// TIA Portal V19 export
DATA_BLOCK "Sys"   // DB10
// stored: Access Published, MemoryReserve 100
   VAR
      Bit1 : Bool;   // Always ON
      Bit0 : Bool;   // Always OFF
      ByPass : Bool;   // Temporary BYPASS
      AuxFirstPLCCycle : Bool;
      FirstPLCCycle : Bool;
      ClockCyc : Bool;
      Clock_250MS : Bool;
      Clock_500MS : Bool;
      Clock_1S : Bool;
      Clock_2S : Bool;
      Clock_4S : Bool;
      Clock_8S : Bool;
      Clock_16S : Bool;
      Clock_32S : Bool;
      Clock_64S : Bool;
      LampTest : Bool;
      LampTestMem : Bool;
      SimulationDevice : Bool;
      PreviousCycleTime : Int;
      OB_82_Execution : Bool;
      OB_83_Execution : Bool;
      OB_86_Execution : Bool;
      OB_122_Execution : Bool;
      OB_121_Execution : Bool;
      "I/O_Missing" : Bool;
   END_VAR
BEGIN
END_DATA_BLOCK
